SUBAPPLICATION Uebung_019b_AX (* Umschalten einer Maske, mit Plug and Socket *)
  (* Standard: 61499-2; Description: Copyright (c) 2026 Meisterschulen am Ostbahnhof This program and the accompanying materials are made available under the terms of the Eclipse Public License 2.0 which is available at https://www.eclipse.org/legal/epl-2.0/ SPDX-License-Identifier: EPL-2.0 *)
  (* Version 1.0, 2026-09-09, Franz Höpfinger, Meisterschulen am Ostbahnhof, initial API and implementation and/or initial documentation *)
  PACKAGE Uebungen;
  IMPORT Uebungen::const::UT::DefaultPool::AlarmMask_A2_medium;
  IMPORT Uebungen::const::UT::DefaultPool::DataMask_M1;
  IMPORT Uebungen::const::UT::DefaultPool::DataMask_M2;
  IMPORT isobus::UT::Q::const::IDs::ID_NULL;
  IMPORT isobus::UT::io::Softkey::SoftKeyActivationCode::SK_PRESSED;
  IMPORT logiBUS::io::DI::logiBUS_DI::Input_I1;
  IMPORT logiBUS::io::DI::logiBUS_DI::Input_I2;
  IMPORT logiBUS::io::DI::logiBUS_DI::Input_I3;
  IMPORT logiBUS::io::DI::logiBUS_DI_Events::BUTTON_SINGLE_CLICK;
  IMPORT logiBUS::io::DQ::logiBUS_DO::Output_Q1;
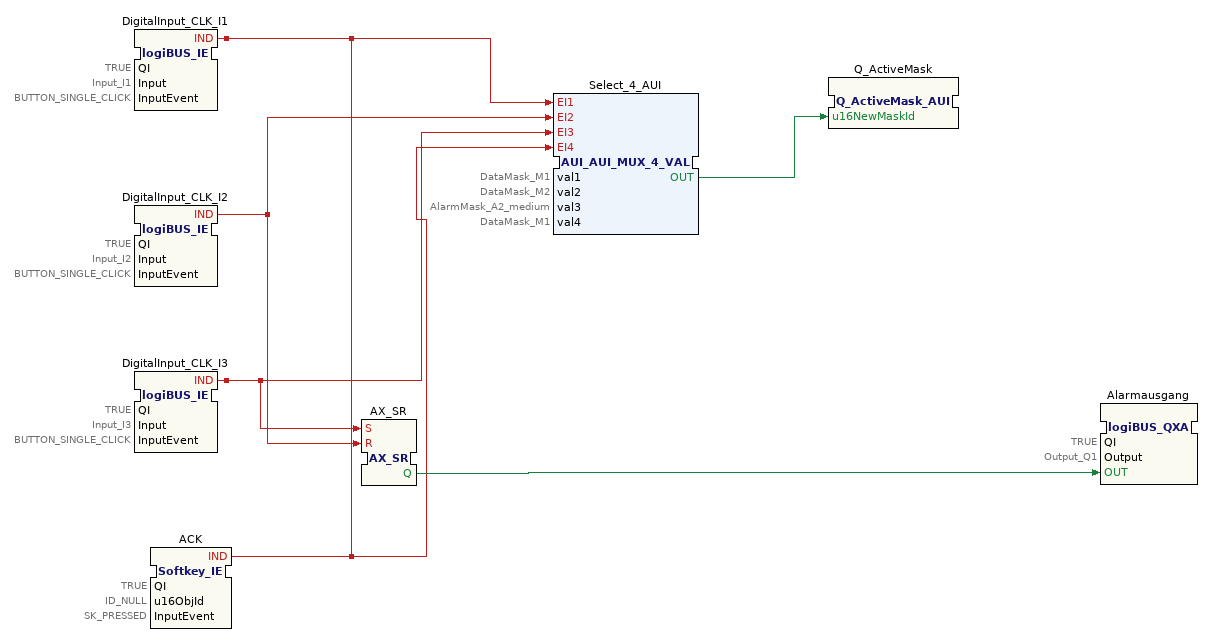
  FBS
    DigitalInput_CLK_I1 : logiBUS::io::DI::logiBUS_IE(QI := TRUE, Input := Input_I1, InputEvent := BUTTON_SINGLE_CLICK);
    DigitalInput_CLK_I2 : logiBUS::io::DI::logiBUS_IE(QI := TRUE, Input := Input_I2, InputEvent := BUTTON_SINGLE_CLICK);
    DigitalInput_CLK_I3 : logiBUS::io::DI::logiBUS_IE(QI := TRUE, Input := Input_I3, InputEvent := BUTTON_SINGLE_CLICK);
    ACK : isobus::UT::io::Softkey::Softkey_IE(QI := TRUE, u16ObjId := ID_NULL, InputEvent := SK_PRESSED);
    Q_ActiveMask : isobus::UT::Q::Q_ActiveMask_AUI;
    AX_SR : adapter::events::unidirectional::AX_SR;
    Alarmausgang : logiBUS::io::DQ::logiBUS_QXA(QI := TRUE, Output := Output_Q1);
  END_FBS
  SUBAPPS
    Select_4_AUI : MyLib::sys::AUI_AUI_MUX_4_VAL(val1 := DataMask_M1, val2 := DataMask_M2, val3 := AlarmMask_A2_medium, val4 := DataMask_M1);
  END_SUBAPPS
  EVENT_CONNECTIONS
    DigitalInput_CLK_I1.IND TO Select_4_AUI.EI1;
    DigitalInput_CLK_I2.IND TO Select_4_AUI.EI2;
    DigitalInput_CLK_I3.IND TO Select_4_AUI.EI3;
    ACK.IND TO Select_4_AUI.EI4;
    DigitalInput_CLK_I3.IND TO AX_SR.S;
    DigitalInput_CLK_I2.IND TO AX_SR.R;
    DigitalInput_CLK_I1.IND TO AX_SR.R;
    ACK.IND TO AX_SR.R;
  END_CONNECTIONS
  ADAPTER_CONNECTIONS
    Select_4_AUI.OUT TO Q_ActiveMask.u16NewMaskId;
    AX_SR.Q TO Alarmausgang.OUT;
  END_CONNECTIONS
END_SUBAPPLICATION
